Omron CX-Programmer project NewProject (CX-Programmer 9.70)

# PLC NewPLC1: CP1E E20

## Global symbols (name address type ; comment)
0.01 BOOL  ; STOP
0.02 BOOL  ; START_1
0.03 BOOL  ; START_2
100.00 BOOL  ; LED_1
100.01 BOOL  ; LED_2

## Program NewProgram1 (cyclic task 0)

### Section Section1

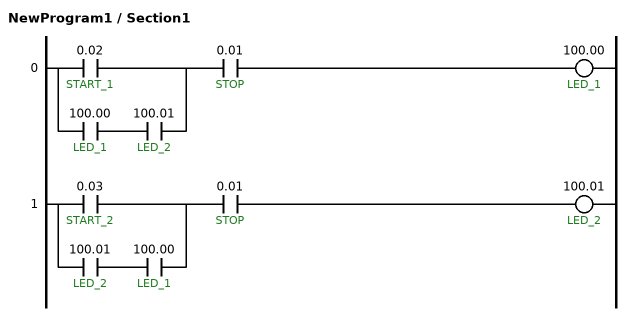
; rung 0
LD 0.02  ; START_1
LD 100.00  ; LED_1
AND 100.01  ; LED_2
ORLD
AND 0.01  ; STOP
OUT 100.00  ; LED_1
; rung 1
LD 0.03  ; START_2
LD 100.01  ; LED_2
AND 100.00  ; LED_1
ORLD
AND 0.01  ; STOP
OUT 100.01  ; LED_2

### Section END
; rung 0
END(001)